PROGRAM MAIN
VAR
	bStart : BOOL;
	
	stBottle1 : ST_Bottle := (nId := 101, fTargetLevel := 70, eLiquidType := E_LiquidType.HONEY);
	stBottle2 : ST_Bottle := (nId := 102, fTargetLevel := 85, eLiquidType := E_LiquidType.SODA);
	stBottle3 : ST_Bottle := (nId := 103, fTargetLevel := 90, eLiquidType := E_LiquidType.WATER);
	
	
	fbStationController1 : FB_StationController;
	fbStationController2: FB_StationController;
	fbStationController3 : FB_StationController;
	
	
END_VAR

IF bStart THEN
	fbStationController1(stBottle := stBottle1);
	fbStationController2(stBottle := stBottle2);
	//fbStationController3(stBottle := stBottle3);
	bStart := FALSE;
END_IF

END_PROGRAM

(* stored: Version 1.1.0.1, ProductVersion 3.1.4024.16
   POU MAIN: Id {503e582f-e132-4453-86b2-ff7b3fc71ee6}, SpecialFunc None *)
